{attribute 'GeneratedUsingTerminal: EJ5151-0000-0016'}
{attribute addProperty BoxType "EJ5151-0000-0016"}
{attribute addProperty Id "Period_valueAT %I*UDINT4"}
{attribute addProperty CRC "615922771"}
{attribute addProperty Size "4"}
TYPE ENC_Inputs_24B63C53 :
STRUCT
	{attribute addProperty Name "Period_value"}
	Period_value AT %I* : UDINT;
END_STRUCT
END_TYPE

(* stored: Version 1.2.0.0, ProductVersion 3.1.4024.9
   DUT ENC_Inputs_24B63C53: Id {8e174ecc-e8d1-4c53-821d-24c5cb99d99e} *)
